// TIA Portal V16 export
// export: Created 2022-09-01T14:29:22.7740587Z, ExportSetting WithDefaults, DisplayName Totally Integrated Automation Portal, DisplayVersion V16, DisplayName TIA Portal Version Control Interface, DisplayVersion V16, DisplayName TIA Portal Openness, DisplayVersion V16, DisplayName STEP 7 Professional, DisplayVersion V16, DisplayName STEP 7 Safety, DisplayVersion V16, DisplayName WinCC Advanced, DisplayVersion V16
FUNCTION "Medidor_Caudal_FQ301" : Void   // FC11, LAD
{ S7_Optimized_Access := 'TRUE' }
VERSION : 0.1
// stored: AutoNumber true, IsIECCheckEnabled false, SetENOAutomatically false, UDAEnableTagReadback false
BEGIN

REGION Network 1
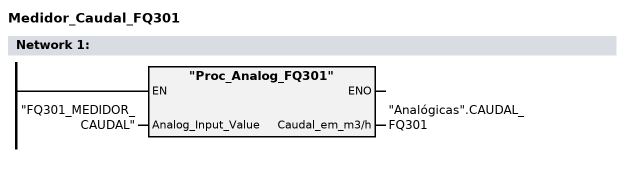
   RUNG wire#powerrail
      "Proc_Analog_FQ301"(Analog_Input_Value := "FQ301_MEDIDOR_CAUDAL", "Caudal_em_m3/h" => "Analógicas".CAUDAL_FQ301)
   END_RUNG
   // the same network as SCL:
   "Proc_Analog_FQ301"(Analog_Input_Value := "FQ301_MEDIDOR_CAUDAL",
                       "Caudal_em_m3/h" => "Analógicas".CAUDAL_FQ301);
END_REGION
END_FUNCTION
